FUNCTION_BLOCK DigitalInput_ForceVisitor_TEST
VAR
END_VAR

ForceOffVisitor_NO();
ForceOnVisitor_NO();
UnforcedVisitor_NO();
ForceOffVisitor_NC();
ForceOnVisitor_NC();
UnforcedVisitor_NC();

METHOD ForceOffVisitor_NC
VAR
	Expected	 : BOOL;
	Actual		 : BOOL;
	Input		 : BOOL;
	DigitalInput : DigitalInput_NC('DigitalInput', Input);
	ForceVisitor : ForceVisitor;
END_VAR
IF TestSuite.Test(__POUNAME()).ExecuteTest() THEN
	Expected		   := FALSE;
	DigitalInput.Force := E_ForceState.ForceOn;
	ForceVisitor.Force := E_ForceState.ForceOff;
	DigitalInput.Accept(ForceVisitor);
	Input  := FALSE;
	Actual := DigitalInput.IsActive;
	TestSuite.Test(__POUNAME()).AssertEqual(Expected, Actual);
END_IF
END_METHOD

METHOD ForceOffVisitor_NO
VAR
	Expected	 : BOOL;
	Actual		 : BOOL;
	Input		 : BOOL;
	DigitalInput : DigitalInput_NO('DigitalInput', Input);
	ForceVisitor : ForceVisitor;
END_VAR
IF TestSuite.Test(__POUNAME()).ExecuteTest() THEN
	Expected		   := FALSE;
	DigitalInput.Force := E_ForceState.ForceOn;
	ForceVisitor.Force := E_ForceState.ForceOff;
	DigitalInput.Accept(ForceVisitor);
	Input  := TRUE;
	Actual := DigitalInput.IsActive;
	TestSuite.Test(__POUNAME()).AssertEqual(Expected, Actual);
END_IF
END_METHOD

METHOD ForceOnVisitor_NC
VAR
	Expected	 : BOOL;
	Actual		 : BOOL;
	Input		 : BOOL;
	DigitalInput : DigitalInput_NC('DigitalInput', Input);
	ForceVisitor : ForceVisitor;
END_VAR
IF TestSuite.Test(__POUNAME()).ExecuteTest() THEN
	Expected		   := TRUE;
	DigitalInput.Force := E_ForceState.ForceOff;
	ForceVisitor.Force := E_ForceState.ForceOn;
	DigitalInput.Accept(ForceVisitor);
	Input  := FALSE;
	Actual := DigitalInput.IsActive;
	TestSuite.Test(__POUNAME()).AssertEqual(Expected, Actual);
END_IF
END_METHOD

METHOD ForceOnVisitor_NO
VAR
	Expected	 : BOOL;
	Actual		 : BOOL;
	Input		 : BOOL;
	DigitalInput : DigitalInput_NO('DigitalInput', Input);
	ForceVisitor : ForceVisitor;
END_VAR
IF TestSuite.Test(__POUNAME()).ExecuteTest() THEN
	Expected		   := TRUE;
	DigitalInput.Force := E_ForceState.ForceOff;
	ForceVisitor.Force := E_ForceState.ForceOn;
	DigitalInput.Accept(ForceVisitor);
	Input  := FALSE;
	Actual := DigitalInput.IsActive;
	TestSuite.Test(__POUNAME()).AssertEqual(Expected, Actual);
END_IF
END_METHOD

METHOD UnforcedVisitor_NC
VAR
	Expected	 : BOOL;
	Actual		 : BOOL;
	Input		 : BOOL;
	DigitalInput : DigitalInput_NC('DigitalInput', Input);
	ForceVisitor : ForceVisitor;
END_VAR
IF TestSuite.Test(__POUNAME()).ExecuteTest() THEN
	Expected		   := TRUE;
	DigitalInput.Force := E_ForceState.ForceOn;
	ForceVisitor.Force := E_ForceState.Unforced;
	DigitalInput.Accept(ForceVisitor);
	Input  := FALSE;
	Actual := DigitalInput.IsActive;
	TestSuite.Test(__POUNAME()).AssertEqual(Expected, Actual);
END_IF
END_METHOD

METHOD UnforcedVisitor_NO
VAR
	Expected	 : BOOL;
	Actual		 : BOOL;
	Input		 : BOOL;
	DigitalInput : DigitalInput_NO('DigitalInput', Input);
	ForceVisitor : ForceVisitor;
END_VAR
IF TestSuite.Test(__POUNAME()).ExecuteTest() THEN
	Expected		   := FALSE;
	DigitalInput.Force := E_ForceState.ForceOn;
	ForceVisitor.Force := E_ForceState.Unforced;
	DigitalInput.Accept(ForceVisitor);
	Input  := FALSE;
	Actual := DigitalInput.IsActive;
	TestSuite.Test(__POUNAME()).AssertEqual(Expected, Actual);
END_IF
END_METHOD

END_FUNCTION_BLOCK

(* stored: Version 1.1.0.1, ProductVersion 3.1.4026.18
   POU DigitalInput_ForceVisitor_TEST: Id {12345678-1234-1234-1234-123456789abc}, SpecialFunc None
   Method ForceOffVisitor_NC: Id {87654321-4321-4321-4321-cba987654321}
   Method ForceOffVisitor_NO: Id {11111111-2222-3333-4444-555555555555}
   Method ForceOnVisitor_NC: Id {aaaaaaaa-bbbb-cccc-dddd-eeeeeeeeeeee}
   Method ForceOnVisitor_NO: Id {22222222-3333-4444-5555-666666666666}
   Method UnforcedVisitor_NC: Id {dddddddd-eeee-ffff-aaaa-bbbbbbbbbbbb}
   Method UnforcedVisitor_NO: Id {33333333-4444-5555-6666-777777777777} *)
